(* IEC 61131-3 sources: AXOpen/src/core/ctrl/src/AxoArrays, 2 files *)

(* ---- AxoBoolArray.st ---- *)
NAMESPACE AXOpen.Core
    {S7.extern=ReadWrite}
    CLASS PUBLIC AxoBoolArray
        VAR PUBLIC
            DataChanged : BOOL;
        END_VAR

        METHOD PUBLIC ToggleDataChangedFlag
            DataChanged := NOT DataChanged;
        END_METHOD

        VAR PRIVATE
            _dataChanged : BOOL;
        END_VAR

        METHOD PUBLIC DataHasChanged: BOOL
            DataHasChanged := DataChanged XOR _dataChanged;
            _dataChanged := DataChanged;
        END_METHOD
    END_CLASS
END_NAMESPACE

(* ---- AxoByteArray.st ---- *)
NAMESPACE AXOpen.Core
    {#ix-prop: public string DisplayFormat}
    {S7.extern=ReadWrite}
    CLASS PUBLIC AxoByteArray
        VAR PUBLIC
            DataChanged : BOOL;
        END_VAR

        METHOD PUBLIC ToggleDataChangedFlag
            DataChanged := NOT DataChanged;
        END_METHOD
    END_CLASS
END_NAMESPACE
